// TIA Portal V16 export
// export: Created 2024-12-03T15:41:45.9214731Z, ExportSetting WithReadOnly, DisplayName Totally Integrated Automation Portal, DisplayVersion V16 Update 6, DisplayName TIA Portal Version Control Interface, DisplayVersion V16 Update 2, DisplayName TIA Portal Openness, DisplayVersion V16 Update 6, DisplayName TIA Portal Teamcenter Gateway, DisplayVersion V16, DisplayName SINAMICS Startdrive Advanced, DisplayVersion V16 Update 5, DisplayName SINAMICS Startdrive G130, G150, S120, S150, SINAMICS MV, S210, DisplayVersion V16 Update 5, DisplayName SINAMICS Startdrive G110M, G120, G120C, G120D, G120P, G115D, DisplayVersion V16 Update 5, DisplayName STEP 7 Professional, DisplayVersion V16 Update 6, DisplayName STEP 7 Safety, DisplayVersion V16, DisplayName WinCC Advanced / Unified PC, DisplayVersion V16 Update 6
TYPE "Counter_UDT"
// stored: CreationDate 2021-07-13T07:41:36.2278727Z, InterfaceModifiedDate 2020-10-03T05:30:31.7241702Z, IsConsistent true, LibraryConformanceStatus The object is library-conformant., ModifiedDate 2021-03-27T07:36:39.8858995Z
   STRUCT
      Cmd : Struct
         CountUp : Bool;
         ShiftHours : Bool;
         Reset : Bool;
      END_STRUCT;
      CounterStatus : Struct
         TotalCounter : UInt;
         HourlyCounters : Array[0..7] of UInt;
         MovingAverageCounters : Array[0..59] of UInt;
         CapacityCounter05Min : UInt;
         CapacityCounter10Min : UInt;
         CapacityCounter15Min : UInt;
      END_STRUCT;
      "Name" : String;
      Zone : UInt;
   END_STRUCT;
END_TYPE
